// TIA Portal V19 export
VAR_GLOBAL   // PLC tag table "IPC_MSG_TOPIC_CONST"
END_VAR
VAR_GLOBAL CONSTANT   // user constants
   LOG_MSG_ITEMS : Int := 5;
   LOG_TOPIC_PAR_CHANGE : UDInt := 1000;
   LOG_TOPIC_InizioSetup : UDInt := 101;
   LOG_TOPIC_FineSetup : UDInt := 102;
END_VAR
